{attribute addProperty BoxType "EK1122-0000-0018"}
{attribute addProperty Id "Beckhoff_EJ7xxxsub_EK1100EK1100_179A0949162"}
{attribute addProperty CRC "580471506"}
{attribute addProperty SizeInBites "16"}
{attribute addProperty SizeInBytes "2"}
TYPE Beckhoff_EJ7xxxEK1122_22994AD2 EXTENDS EK1122_179A0949 :
STRUCT
	{attribute addProperty Name "Beckhoff_EJ7xxxsub_EK1100"}
	Beckhoff_EJ7xxxsub_EK1100 : EK1100_179A0949;
END_STRUCT
END_TYPE

(* stored: Version 1.2.0.0, ProductVersion 3.1.4024.9
   DUT Beckhoff_EJ7xxxEK1122_22994AD2: Id {edb9aa61-4260-4a79-af19-61a48a88d2f0} *)
